FUNCTION_BLOCK EnableGroup  IMPLEMENTS I_Task
VAR
	groupEnable			: MC_GroupEnable;
	_caGroup			: I_CollisionGroup;
	_Done 				: BOOL;
	_Error				: BOOL;
	_ErrorID			: UDINT;
END_VAR

{analysis -2}

METHOD Abort : BOOL
groupEnable.Execute := FALSE;
Abort := TRUE;
END_METHOD

PROPERTY Busy : BOOL
GET
Busy := groupEnable.Busy;
END_GET
END_PROPERTY

METHOD Cycle : HRESULT
VAR_INPUT
END_VAR
IF _caGroup = 0 THEN
	cycle := -1;
	RETURN;
END_IF
_Done := groupEnable.Done OR _Done;
_Error := groupEnable.Error OR _Error;
IF groupEnable.ErrorId <> 0 THEN
	_ErrorId := groupEnable.ErrorId;
END_IF
groupEnable(AxesGroup := _caGroup.GroupRef);
groupEnable.Execute := FALSE;
END_METHOD

PROPERTY Done : BOOL
GET
Done := _Done;
END_GET
END_PROPERTY

PROPERTY Error : BOOL
GET
Error := _Error;
END_GET
END_PROPERTY

METHOD Execute : HRESULT
IF groupEnable.Execute THEN
	Execute := -1;
	RETURN;
END_IF

IF _caGroup = 0 THEN
	Execute := -2;
	RETURN;
END_IF

groupEnable.Execute := TRUE;
END_METHOD

PROPERTY MyCollisionGroup : I_CollisionGroup
GET
MyCollisionGroup := _caGroup;
END_GET
SET
IF MyCollisionGroup <> 0 THEN
	_caGroup := MyCollisionGroup;
END_IF
END_SET
END_PROPERTY

END_FUNCTION_BLOCK

(* stored: Version 1.1.0.1
   POU EnableGroup: Id {01c66182-3535-4445-8b1b-a8f549e6d0ab}, SpecialFunc None
   Method Abort: Id {8e535bd0-5fdc-4fa1-a309-8fd0da8ee400}
   Property Busy: Id {4e4db787-2247-4ffa-a4fa-212f7c481400}
   Get Get: Id {8a7815a8-c1fd-47de-9b79-1b1569675505}
   Method Cycle: Id {53999691-fece-418c-ba0c-d2348e6bf666}
   Property Done: Id {a772c0a8-091e-4c87-9bf2-8f9e57381133}
   Get Get: Id {50223277-a964-4c91-8fe3-3b1b9979de48}
   Property Error: Id {3c7c1991-df63-4a12-9a6d-e45eb55d1f39}
   Get Get: Id {f9f90eb7-811c-45c6-9af2-24f6616a22a6}
   Method Execute: Id {6b5a42b1-94d9-46bc-bf55-d1fbc24c1815}
   Property MyCollisionGroup: Id {4ec7cc23-7094-408b-87af-591e7c9596ca}
   Get Get: Id {7e162f97-609a-4d5e-8ef7-d97f2590a7d7}
   Set Set: Id {f6b98b9b-247c-45c3-9781-3be9ceb23789} *)
